FUNCTION_BLOCK FB_VisuControlHmi
VAR_INPUT
END_VAR
VAR_OUTPUT
END_VAR

mTcHmiDebug();
mComboBox();
mValveMaskEntry();

METHOD mComboBox
VAR
	aTexts : ARRAY [1..3] OF STRING := ['Decimal','Binary','Hex'];
	bIni: BOOL := TRUE;
	nCounter: INT := 3;
END_VAR
// set the Combobox entries in the first cycle
IF bIni THEN
	FOR nCounter := 1 TO 3 DO
		GVL_VisuControlHMI.aComboboxEntries[nCounter].id := nCounter;
		GVL_VisuControlHMI.aComboboxEntries[nCounter].text := CONCAT('Display', aTexts[nCounter]);
		GVL_VisuControlHMI.aComboboxEntries[nCounter].value := nCounter * 10;
	END_FOR

	bIni := FALSE;
END_IF
END_METHOD

METHOD mDisplayFormat : STRING
VAR_INPUT
	nValue      : DWORD;   // Value to display
END_VAR
VAR
    eFormat     : INT; // Selected format
    nBitWidth   : INT := 16; // For binary (8,16,32)
    sOut        : STRING(50); // Output for Visu binding
END_VAR
eFormat := GVL_VisuControlHMI.nSelectedValue;
CASE eFormat OF

    E_DisplayFormat.Decimal:
        sOut := DWORD_TO_STRING(nValue);

    E_DisplayFormat.Binary:
        sOut := DWORD_TO_BINSTR(nValue, nBitWidth);

    E_DisplayFormat.Hex:
        sOut := DWORD_TO_HEXSTR(nValue, (nBitWidth / 4), FALSE);

END_CASE

mDisplayFormat := sOut;
END_METHOD

METHOD mTcHmiDebug
VAR_INPUT
END_VAR
END_METHOD

METHOD mValveMaskEntry
VAR_INPUT
END_VAR
VAR
	Idx : UINT;
END_VAR
Idx := GVL_VisuControlHMI.visValveMaskIdx;

	IF GVL_VisuControlHMI.nValveMask <> 0 THEN
		GVL_VisuControlHMI.anValveMaskListToRecipe[Idx] := GVL_VisuControlHMI.nValveMask;
		GVL_VisuControlHMI.nValveMask := 0; // To Clear the Text Box
		GVL_VisuControlHMI.anValveMaskListToDisplay[Idx] := mDisplayFormat(nValue := GVL_VisuControlHMI.nValveMask) ;
	END_IF
END_METHOD

END_FUNCTION_BLOCK

(* stored: Version 1.1.0.1
   POU FB_VisuControlHmi: Id {44e419da-d1ca-0ad4-1138-0ce61d4d2251}, SpecialFunc None
   Method mComboBox: Id {3f7fceb7-e492-065f-2216-b4ade514c6de}
   Method mDisplayFormat: Id {1f6273d3-5414-06ca-0b15-14107082be32}
   Method mTcHmiDebug: Id {b41e4dad-3992-0a34-2486-613cd7bbc33c}
   Method mValveMaskEntry: Id {0ec0a1ee-16c0-0ede-223e-2794791150b7} *)
